(* IEC 61131-3 sources: volt/packages/volt-lsp-iec/test-corpus/lenze-mid/Device/Plc Logic/Application/MotionControl, 2 files *)

(* ---- Mach1_MotionControl.pou ---- *)
PROGRAM Mach1_MotionControl
VAR
//Main Cabinet
	Maindrive: Camming;
	WrappingDevice: Camming;
	Sidecorrection: Camming_SideCorrection;
	Fan: ATD_FQI;
	Bobbin: ATD_TorqueControl;

//ATF
	FeedForwardADS: ATD_FQI;
	FeedForwardATF: ATD_FQI;
	Elevator: ATD_FQI;

	FeedForwardWrapper: BasicMovement;
	VirtualMaster_0: VirtualMaster;
	identPolePosition_FeedforwardWrapper: identPolePosition;
	L_MC1P_ChangeMachineData_MainDrive: L_MC1P_ChangeMachineData;
	xMainDriveDoneOnce: BOOL;
	xFeedforwardDoneOnce: BOOL;
	xWrappingDeviceDoneOnce: BOOL;
	L_MC1P_ChangeMachineData_FeedforwardWrapper: L_MC1P_ChangeMachineData;
	L_MC1P_ChangeMachineData_WrappingDevice: L_MC1P_ChangeMachineData;
END_VAR

%LANGUAGE LD
%NETWORK
VirtualMaster_0(ioDataExchange := Data_Exchange_Motion.Servo_VirtualMaster, i_xPositionIsRetain := TRUE, i_lrWindowStandstill := 1, i_lrJogVel := 5, i_VelMax := 600, ioSlaveAxis := LM_VirtualMaster);
%NETWORK
ASSIGN(L_MC1P_ChangeMachineData_MainDrive(Axis := Axis_MainDrive, xExecute := Axis_MainDrive.xCommunicationOK AND INVERT(Axis_MainDrive.xDriveEnabled), xSetOrientation := TRUE, xOrientation := LST_InputsOutputs.I100_5_ConfigSelectionRightMachine), Q_SET => xMainDriveDoneOnce);
%NETWORK
ASSIGN(Data_Exchange_Motion.Servo_MainDrive.Control.Enable AND xMainDriveDoneOnce, Q => Data_Exchange_Motion.Servo_MainDrive.Control.Enable);
%NETWORK "Main drive motion"
Maindrive(EN := RAIL(), ioDataExchange := Data_Exchange_Motion.Servo_MainDrive, i_xOnlyPositiveDirectionSync := TRUE, i_lrWindowStandstill := 1, i_lrJogVel := 2, i_lrSyncVel := 10, i_CamCyclic := TRUE, i_MasterAbsolute := TRUE, i_SlaveAbsolute := TRUE, ioMasterAxis := LM_VirtualMaster, ioSlaveAxis := Axis_MainDrive);
%NETWORK
ASSIGN(L_MC1P_ChangeMachineData_WrappingDevice(Axis := Axis_OverrollingDevice, xExecute := Axis_OverrollingDevice.xCommunicationOK AND INVERT(Axis_OverrollingDevice.xDriveEnabled), xSetOrientation := TRUE, xOrientation := INVERT(LST_InputsOutputs.I100_5_ConfigSelectionRightMachine)), Q_SET => xWrappingDeviceDoneOnce);
%NETWORK
ASSIGN(Data_Exchange_Motion.Servo_WrappingDevice.Control.Enable AND xWrappingDeviceDoneOnce, Q => Data_Exchange_Motion.Servo_WrappingDevice.Control.Enable);
%NETWORK "Wrapping device"
WrappingDevice(EN := RAIL(), ioDataExchange := Data_Exchange_Motion.Servo_WrappingDevice, i_xOnlyPositiveDirectionSync := FALSE, i_lrWindowStandstill := 5, i_lrJogVel := 10, i_lrSyncVel := 10, i_CamCyclic := TRUE, i_MasterAbsolute := TRUE, i_SlaveAbsolute := FALSE, ioMasterAxis := LM_VirtualMaster, ioSlaveAxis := Axis_OverrollingDevice);
%NETWORK "Side correction"
Sidecorrection(EN := RAIL(), ioDataExchange := Data_Exchange_Motion.Servo_SideCorrection, i_xOnlyPositiveDirectionSync := FALSE, i_lrWindowStandstill := 5, i_lrJogVel := 100, i_lrSyncVel := 10, i_CamCyclic := TRUE, i_MasterAbsolute := TRUE, i_SlaveAbsolute := FALSE, ioMasterAxis := LM_VirtualMaster, ioSlaveAxis := Axis_SideCorrection);
%NETWORK
ASSIGN(L_MC1P_ChangeMachineData_FeedforwardWrapper(Axis := Axis_FeedFowardWrapper, xExecute := Axis_FeedFowardWrapper.xCommunicationOK AND INVERT(Axis_FeedFowardWrapper.xDriveEnabled), xSetOrientation := TRUE, xOrientation := LST_InputsOutputs.I100_5_ConfigSelectionRightMachine), Q_SET => xFeedforwardDoneOnce);
%NETWORK
identPolePosition_FeedforwardWrapper(execute := AND(xFeedforwardDoneOnce, Axis_FeedFowardWrapper.xCommunicationOK, INVERT(Axis_FeedFowardWrapper.xSTOActive)), ioAxis := Axis_FeedFowardWrapper);
%NETWORK
ASSIGN(Data_Exchange_Motion.FeedForwardWrapper.Control.Enable AND identPolePosition_FeedforwardWrapper.doneOnce, Q => Data_Exchange_Motion.FeedForwardWrapper.Control.Enable);
%NETWORK "Feed forward wrapper DTA"
FeedForwardWrapper(ioDataExchange := Data_Exchange_Motion.FeedForwardWrapper, TouchProbeSensor := INVERT(LST_InputsOutputs.I101_0_Wrapper_present), i_lrWindowStandstill := 5, i_lrJogVel := 10, ioSlaveAxis := Axis_FeedFowardWrapper);
%NETWORK "FQI Bobbin"
Bobbin(lrAcc := 6000, lrDec := 6000, ioAxis := Axis_Bobbin, DataIO := Data_Exchange_Motion.FQI_Bobbin, lrTorque := Data_Exchange_Motion.BobbinTorque);
%NETWORK "FQI Fan"
Fan(lrAcc := 500, lrDec := 75, ioAxis := Axis_Fan, DataIO := Data_Exchange_Motion.FQI_Fan);
%NETWORK "FQI FeedForward ADS"
FeedForwardADS(lrAcc := 6000, lrDec := 6000, ioAxis := Axis_FeedForwardADS, DataIO := Data_Exchange_Motion.FQI_FeedforwardADS);
%NETWORK "FQI FeedForward  ATF"
FeedForwardATF(lrAcc := 6000, lrDec := 1500, ioAxis := Axis_FeedForwardATF, DataIO := Data_Exchange_Motion.FQI_FeedforwardATF);
%NETWORK "FQI Elevator"
Elevator(lrAcc := 50, lrDec := 200, ioAxis := Axis_Elevator, DataIO := Data_Exchange_Motion.FQI_ElevatorATF);

END_PROGRAM

(* ---- POU.pou ---- *)
PROGRAM POU
VAR
	L_TS2P_FlexCamState_0: L_TS2P_FlexCamState;
END_VAR

%LANGUAGE FBD
%NETWORK
L_TS2P_FlexCamState_0();
%NETWORK
L_MC1P_AxisBasicControlV2();
%NETWORK
L_TT1P_BasicMotionBase();
%NETWORK
L_TT1P_FlexCamBase();
%NETWORK
L_TT1P_FlexCamState();

END_PROGRAM
